(* CODESYS project em_log_test.project

Project tree, tasks and I/O mapping:
  Device : EMICON-ARM Cortex-A8-Linux, EMICON, version 3.5.17.20
      settings: IP = '192.168.0.50'; Emicon settings version = '0.0.2.0'
    application Application
      libraries: Standard, * (System); CmpErrors Interfaces, * (System); CmpApp, 3.5.17.0 (System); EmiconLog, 3.5.17.20 (Emicon)
      task MainTask (cyclic, interval t#500ms, priority 1) calls PLC_PRG
      program PLC_PRG [ST]
      global variables GVL
*)

// Device/Application/GVL
VAR_GLOBAL CONSTANT
	OWN_EVENT_ID_CLR: BYTE := 0;
	OWN_EVENT_ID_STOP: BYTE := 1;
	OWN_EVENT_ID_START: BYTE := 2;
	OWN_EVENT_CLASS_SYS: BYTE := 0;
	SEVERITY_INFO: BYTE := 6;
END_VAR

// Device/Application/PLC_PRG
PROGRAM PLC_PRG
VAR
	frame_ti1: ARRAY [1..15] OF BYTE := [16#0,16#0,16#0, 16#0,16#0,16#0,16#0, 16#80, 16#CA,16#1B,16#A6,16#14,16#99,16#08,16#10];
	frame_ti2: ARRAY [1..15] OF BYTE := [16#1,16#0,16#0, 16#0,16#0,16#0,16#0, 16#80, 16#CA,16#1B,16#A6,16#14,16#99,16#08,16#10];
	frame_ts1: ARRAY [1..11] OF BYTE := [16#58,16#0,16#0, 16#80, 16#CA,16#1B,16#A6,16#14,16#99,16#08,16#10];
	frame_ts2: ARRAY [1..11] OF BYTE := [16#59,16#0,16#0, 16#80, 16#CA,16#1B,16#A6,16#14,16#99,16#08,16#10];

	i: INT := 1;
	init: BOOL;
END_VAR

IF NOT init THEN
	EmLog.clr_sys_log();
	EmLog.write_sys_log(bySeverity := SEVERITY_INFO, byClassId := OWN_EVENT_CLASS_SYS, byEvent:= 31, dwArgs := 16#00000000);
		// {"class":101, "event":0, "text":"[      ] Конфигурационный файл - %s", "argToInsert":[0,1]},
	EmLog.write_sys_log(bySeverity := SEVERITY_INFO, byClassId := 101, byEvent:= 0, dwArgs := 16#04030200); //{"insert":0, "text":"On"}
		//{"class":102, "event":0, "text":"[0x%04x] Попытка дополнить заполненный буфер", "arg":[0,2]},
	EmLog.write_sys_log(bySeverity := SEVERITY_INFO, byClassId := 102, byEvent:= 0, dwArgs := 16#04030201); // arg = 0x0201
    	//{"class":106, "event":0, "text":"[      ] 'debug_telecontrol' - %s", "argToInsert":[0,1]},
	EmLog.write_sys_log(bySeverity := SEVERITY_INFO, byClassId := 106, byEvent:= 0, dwArgs := 16#04030201);//{"insert":1, "text":"Off"}
    	//{"class":109, "event":0, "text":"[0x%04x] Неработоспособный сокет", "arg":[0,2]},
	EmLog.write_sys_log(bySeverity := SEVERITY_INFO, byClassId := 109, byEvent:= 0, dwArgs := 16#04030201);//arg = 0x0201
    	//{"class":109, "event":1, "text":"[0x%04x] Нарушенная последовательность APDU", "arg":[0,2]},
	EmLog.write_sys_log(bySeverity := SEVERITY_INFO, byClassId := 109, byEvent:= 1, dwArgs := 16#04030201);//arg = 0x0201
    	//{"class":109, "event":2, "text":"[0x%04x] Сработал таймер 1", "arg":[0,2]},
	EmLog.write_sys_log(bySeverity := SEVERITY_INFO, byClassId := 109, byEvent:= 2, dwArgs := 16#04030201);//arg = 0x0201
       // {"class":109, "event":3, "text":"[0x%04x] Неадекватный APCI", "arg":[0,2]},
	EmLog.write_sys_log(bySeverity := SEVERITY_INFO, byClassId := 109, byEvent:= 3, dwArgs := 16#04030201);//arg = 0x0201
        //{"class":109, "event":4, "text":"[0x%04x] Неправильный стартовый символ APDU", "arg":[0,2]},
	EmLog.write_sys_log(bySeverity := SEVERITY_INFO, byClassId := 109, byEvent:= 4, dwArgs := 16#04030201);//arg = 0x0201
        //{"class":109, "event":5, "text":"[0x%04x] Неправильная длина APDU", "arg":[0,2]},
	EmLog.write_sys_log(bySeverity := SEVERITY_INFO, byClassId := 109, byEvent:= 5, dwArgs := 16#04030201);//arg = 0x0201
        //{"class":109, "event":6, "text":"[0x%04x] Отправлен APDU", "arg":[0,2]},
	EmLog.write_sys_log(bySeverity := SEVERITY_INFO, byClassId := 109, byEvent:= 6, dwArgs := 16#04030201);//arg = 0x0201
        //{"class":109, "event":7, "text":"         Формат I (%d,%d)", "arg":[0,2], "arg":[2,2]},
	EmLog.write_sys_log(bySeverity := SEVERITY_INFO, byClassId := 109, byEvent:= 7, dwArgs := 16#04030201);//arg1 = 513 arg2 = 1027
       // {"class":112, "event":0, "text":"[0x%04x] Неудачная попытка создать соединение", "arg":[0,2]},
	EmLog.write_sys_log(bySeverity := SEVERITY_INFO, byClassId := 112, byEvent:= 0, dwArgs := 16#04030201);//arg = 0x0201
        //{"class":112, "event":1, "text":"[0x%04x] Запрос на установление соединения"},												??????
	EmLog.write_sys_log(bySeverity := SEVERITY_INFO, byClassId := 112, byEvent:= 1, dwArgs := 16#04030201);//arg = 0x0201
        //{"class":112, "event":2, "text":"[0x%04x] Установлено соединение c ПУ [0x%04x]", "arg":[0,2], "arg":[2,2]},
	EmLog.write_sys_log(bySeverity := SEVERITY_INFO, byClassId := 112, byEvent:= 2, dwArgs := 16#04030201);//arg1 = 513 arg2 = 1027
       // {"class":112, "event":3, "text":"[0x%04x] Разорвано соединение c ПУ [0x%04x]", "arg":[2,2], "arg":[2,2]},						??????
 	EmLog.write_sys_log(bySeverity := SEVERITY_INFO, byClassId := 112, byEvent:= 3, dwArgs := 16#04030201);//arg1 = 513 arg2 = 1027
      //  {"class":114, "event":0, "text":"%s [0x%04x] Неудачная инициализация", "argToClass":[0,1], "arg":[1,2]},
	EmLog.write_sys_log(bySeverity := SEVERITY_INFO, byClassId := 114, byEvent:= 0, dwArgs := 16#04030264); //class:100, "text":"[App], arg = 0x302
       // {"class":114, "event":1, "text":"%s [0x%04x] Неудачная итерация", "argToClass":[0,1], "arg":[1,2]},
	EmLog.write_sys_log(bySeverity := SEVERITY_INFO, byClassId := 114, byEvent:= 1, dwArgs := 16#04030265); //class:101, "text":"[CfgReader], arg = 0x302
      //  {"class":114, "event":2, "text":"%s [0x%04x] Непредвиденная ситуация - %d", "argToClass":[0,1], "arg":[1,2], "arg":[3,1]},
	EmLog.write_sys_log(bySeverity := SEVERITY_INFO, byClassId := 114, byEvent:= 2, dwArgs := 16#04030266); //"class":102, "text":"[CmdQueue], arg = 0x302, arg = 4
       // {"class":114, "event":3, "text":"%s [0x%04x] Успешная инициализация", "argToClass":[0,1], "arg":[1,2]},
	EmLog.write_sys_log(bySeverity := SEVERITY_INFO, byClassId := 114, byEvent:= 3, dwArgs := 16#04030267); //class:103, "text":"[Connection], arg = 0x302
      //  {"class":114, "event":4, "text":"         Некорректное событие: class - %s, event - %d", "argToClass":[0,1], "arg":[1,1]},
	EmLog.write_sys_log(bySeverity := SEVERITY_INFO, byClassId := 114, byEvent:= 4, dwArgs := 16#04030268); //class:104, "text":"[ControlStat]
       // {"class":114, "event":5, "text":"         IP - %d.%d.%d.%d", "arg":[0,1], "arg":[1,1], "arg":[2,1], "arg":[3,1]},
	EmLog.write_sys_log(bySeverity := SEVERITY_INFO, byClassId := 114, byEvent:= 5, dwArgs := 16#04030201); 
       // {"class":114, "event":6, "text":"%s [0x%04x] Дин.память - %s", "argToClass":[0,1], "arg":[1,2], "argToInsert":[3,1]},
	EmLog.write_sys_log(bySeverity := SEVERITY_INFO, byClassId := 114, byEvent:= 6, dwArgs := 16#04030269); //class":104, "text":"[ControlStat], 0302, Выделение
       // {"class":114, "event":7, "text":"         MemAlloc 0x%08x", "arg":[0,4]},
	EmLog.write_sys_log(bySeverity := SEVERITY_INFO, byClassId := 114, byEvent:= 7, dwArgs := 16#04030201);
       // {"class":114, "event":8, "text":"         MemFree 0x%08x", "arg":[0,4]},
	EmLog.write_sys_log(bySeverity := SEVERITY_INFO, byClassId := 114, byEvent:= 8, dwArgs := 16#04030201);
       // {"class":114, "event":9, "text":"         %s %s [0x%04x]", "argToInsert":[0,1], "argToClass":[1,1], "arg":[2,2]},
	EmLog.write_sys_log(bySeverity := SEVERITY_INFO, byClassId := 114, byEvent:= 9, dwArgs := 16#04036A01); //off , Debug, 0403
       // {"class":115, "event":0, "text":"[      ] Таймаут синхронизации"},
	EmLog.write_sys_log(bySeverity := SEVERITY_INFO, byClassId := 115, byEvent:= 0, dwArgs := 16#04030201);
       // {"class":115, "event":1, "text":"[      ] Обновлено системное время от источника [0x%04x]", "arg":[0,2]},
	EmLog.write_sys_log(bySeverity := SEVERITY_INFO, byClassId := 115, byEvent:= 1, dwArgs := 16#04030201); //0201
       // {"class":116, "event":0, "text":"[      ] Уровень журналирования - %s", "argToSeverity":[0,1]},
	EmLog.write_sys_log(bySeverity := SEVERITY_INFO, byClassId := 116, byEvent:= 0, dwArgs := 16#04030201); //ALERT
       // {"class":118, "event":0, "text":"[0x%04x] Таймаут синхронизации", "arg":[0,2]},
	EmLog.write_sys_log(bySeverity := SEVERITY_INFO, byClassId := 118, byEvent:= 0, dwArgs := 16#04030201); //0201
       // {"class":118, "event":1, "text":"[0x%04x] Получено синхр. время", "arg":[0,2]},
	EmLog.write_sys_log(bySeverity := SEVERITY_INFO, byClassId := 118, byEvent:= 1, dwArgs := 16#04030201); //0201

(*	EmLog.write_ts_log(3, ADR(frame_ts1[1]));
	EmLog.write_ti_log(45, ADR(frame_ti2[1]));
	EmLog.write_ts_log(2, ADR(frame_ts2[1]));
	EmLog.write_ti_log(45, ADR(frame_ti2[1]));
	*)
	EmLog.create_log_files();
	
	init := TRUE;
END_IF

//WHILE EmLog.get_next_log_item(FALSE, ADR(log_str[i])) <> 0 DO
//	i := SEL(i = 100, i + 1, 100);
//END_WHILE

END_PROGRAM
